FUNCTION_BLOCK FbEdgeNeg (* Детектор ниспадающего фронта (среза). *)
  (* Standard: 61499-1; Description: Детектор ниспадающего фронта (среза). Simple FB with one algorithm *)
  (* Version 2.1, 2026-03-20, VA, LIB_PLC *)
  (* Documentation:
  // Детектор ниспадающего фронта (среза). //       DbEdgeNeg //     +-----------+ //     | FbEdgeNeg | //  ->-|In      Out|->- //     +-----------+
  *)
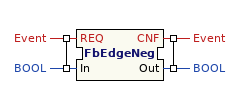
  EVENT_INPUT
    REQ WITH In; (* Normal Execution Request *)
  END_EVENT
  EVENT_OUTPUT
    CNF WITH Out; (* Execution Confirmation *)
  END_EVENT
  VAR_INPUT
    In : BOOL := FALSE; (* Вход. *)
  END_VAR
  VAR_OUTPUT
    Out : BOOL := FALSE; (* Выход. *)
  END_VAR
  VAR
    In_previos : BOOL := FALSE; (* Предыдущее состояние входа. *)
  END_VAR
  EC_STATES
    REQ : REQ -> CNF;
  END_STATES
  ALGORITHM REQ IN ST:
// Детектор ниспадающего фронта (среза).
Out := In_previos AND NOT (In);
// Запомнить предыдущее состояние входа.
In_previos := In;

// @COPYLEFT ALL WRONGS RESERVED :)
// Author: VA
// Contacts: DIY.PLC.314@gmail.com
// Date start LIB_PLC: 2014
// License: GNU GPL-2.0-or-later
// https://www.gnu.org/licenses/old-licenses/gpl-2.0.html
// https://www.youtube.com/watch?v=n1F_MfLRlX0
// https://www.youtube.com/@DIY_PLC
// https://github.com/DIYPLC/LIB_PLC
// https://oshwlab.com/diy.plc.314/PLC_HW1_SW1
// https://3dtoday.ru/3d-models/mechanical-parts/body/korpus-na-din-reiku
// https://t.me/DIY_PLC
  END_ALGORITHM
END_FUNCTION_BLOCK
